{attribute 'GeneratedUsingTerminal: EK1960-2600-0019'}
{attribute addProperty BoxType "EK1960-2600-0019"}
{attribute addProperty Id "FSOEAT %I*FSOE_BAA7477B48"}
{attribute addProperty CRC "2421954868"}
{attribute addProperty Size "48"}
TYPE FSoE_Inputs_905C1934 :
STRUCT
	{attribute addProperty Name "FSOE"}
	FSOE AT %I* : FSOE_BAA7477B;
END_STRUCT
END_TYPE

(* stored: Version 1.2.0.0, ProductVersion 3.1.4024.9
   DUT FSoE_Inputs_905C1934: Id {f2e81307-1c29-4ae9-add8-e8a0f4cd6b35} *)
